FUNCTION_BLOCK "SendRcv_iJaw_1TE"   // FB4, SCL
TITLE = SendRcv_iJaw
{ S7_Optimized_Access := 'TRUE' }
AUTHOR : HeitecAg
VERSION : 0.1
// Kommunikation mit den iJaw Backen mittels IO-LInk und Profinet
   VAR_INPUT
      iLADDR_TigoMaster : HW_DEVICE;   // HW-Device aus Hardwarekonfiguration TigoMaster
      iPN_Act : Bool;   // De-/Aktivierung Profinetteilnehmer 1= Aktivieren 0= Deaktivieren
      iCpuRestart : Bool;   // Restartmerker der SPS Wenn keiner vorhanden dann mit False besetzten.
      iAck_Fehler_IoLinkKom : Bool;   // Quitterung des Kommunikationsfehlers.(Sende-/ Lese Aufträge werden danach erneut gestartet)
      iResetIoLinkKom : Bool;   // Reset der LIO-Link kommunikation (Alle Sende-/ Lese Aufträge werden gelöscht)
      iTime_PnIoRyd : Time;   // Zeit zum Hochlauf des Bussystems / des TigoMasters (Vermeidung von Lesefehlern)
      iIJawAktiv_iJaw1 : Bool;   // iJaw 1 ist aktiv & vorhanden
      iIJawAktiv_iJaw2 : Bool;   // iJaw 2 ist aktiv & vorhanden
      iIJawAktiv_iJaw3 : Bool;   // iJaw 3 ist aktiv & vorhanden
      iIJawAktiv_iJaw4 : Bool;   // iJaw 4 ist aktiv & vorhanden
      iFreeIsduCmd : "UDT_iJawISDUCmdData";   // Freier ISDU-Auftrag
      iFreeIsduSendData : Array[0..#LAENGE_IOLINK_RECORD] of Byte;   // Datenbereich zum Schreiben für den freien ISDU-Auftrag
      iUserDaten_iJaw1 : "UDT_iJawDataSendUser";   // Sendedaten PLC --> iJaw 01
      iUserDaten_iJaw2 : "UDT_iJawDataSendUser";   // Sendedaten PLC --> iJaw 02
      iUserDaten_iJaw3 : "UDT_iJawDataSendUser";   // Sendedaten PLC --> iJaw 03
      iUserDaten_iJaw4 : "UDT_iJawDataSendUser";   // Sendedaten PLC --> iJaw 04
   END_VAR
   VAR_OUTPUT
      oError : Bool;   // Fehler bei der Abarbeitung des Bausteines
      oPnTeilAkt : Bool;   // Status des Profinetteilnehmer 1= Teilnehmer aktiv 0= Teilnehmer deaktiviert
      oIoLinkRdy : Bool;   // Ío link kommunikation bereit zum senden / empfangen
      oIoLinkBusy : Bool;   // Ío link kommunikation beschäftig
      oIoLinkError : Bool;   // Ío link kommunikation fehlerhaft
      oFreeIsduCmdFertig : Bool;   // Freier ISDU-Auftrag erfolgreich abgeschlossen
      oFreeIsduCmdDataBereit : Bool;   // Empfange ISDU-Daten liegen bereit
      oFreeIsduRcvData : Array[0..#LAENGE_IOLINK_RECORD] of Byte;   // Empfange ISDU-Daten
      oUserDaten_iJaw1 : "UDT_iJawDataRcvUser";   // Empfangsdaten PLC <-- iJaw 01
      oUserDaten_iJaw2 : "UDT_iJawDataRcvUser";   // Empfangsdaten PLC <-- iJaw 02
      oUserDaten_iJaw3 : "UDT_iJawDataRcvUser";   // Empfangsdaten PLC <-- iJaw 03
      oUserDaten_iJaw4 : "UDT_iJawDataRcvUser";   // Empfangsdaten PLC <-- iJaw 04
   END_VAR
   VAR
      xlocalInit : Bool := TRUE;   // lokale initalisierung
      xlocalError : Bool;   // lokale Fehler ist aufgetreten
      xMin1iJawVorh : Bool;   // mindesten eine iJaw konfiguriert
      xSchrittketteTimeOut : Bool;   // schrittkette hat ein timeout fehler
      xSchrittErsterZyklus : Bool;   // flanke erster zyklus im schritt
      xFehlerSchrittZeitUeberwachung : Bool;   // fehler schrittzeitüberwachung
      xlocalIoLinkRdy : Bool;   // Ío link kommunikation bereit zum senden / empfangen
      xlocalIoLinkBusy : Bool;   // Ío link kommunikation beschäftig
      xlocalIoLinkError : Bool;   // Ío link kommunikation fehlerhaft
      xlocalFreeIsduCmdFertig : Bool;   // Freier ISDU-Auftrag erfolgreich abgeschlossen
      xlocalFreeIsduCmdDataBereit : Bool;   // Empfange ISDU-Daten liegen bereit
      dtCpuSystemDatumZeit : Date_And_Time;   // datum und uhrzeit cpu
      todCpuSystemZeit : Time_Of_Day;   // zeit des tages cpu
      tSchrittZeitVortag : Time;   // schrittzeit vom vortag
      tCpuSystemZeit : Time;   // zeit der cpu
      tStartZeitSchritt : Time;   // startzeit des aktuellen schrittes
      tAktuelleSchrittzeit : Time;   // aktuelle schrittzeit
      tMinSchrittZeit : Time;   // minimum zeit des aktiven schrittes
      tMaxSchrittZeit : Time;   // maximum zeit des aktiven schrittes (T#0ms = schrittzeit überwachung deaktiviert)
      fpCpuRestart : R_TRIG;   // flanke positiv cpu wurde neugestartet
      fpResetIoLink : R_TRIG;   // flanke positiv trigger reset io-link kommunikation / löschen desfifo puffers
      fpPnIOAktiv : R_TRIG;   // flanke positiv profinetteilnehmer ist aktiviert
      fpPnIOInAktiv : R_TRIG;   // flanke positiv profinetteilnehmer ist deaktiviert
      arrIJawVorhandenAktiv : Array[1..#MAX_ANZAHL_IJAWS] of Bool;   // speicher der überprüfung von vorhandenen und aktiven iJaws
      iRetRcvData : Int;   // retval Profinetdaten lesen
      iRetSer : Int;   // retval Profinetdaten umladen
      iRetSendData : Int;   // retval Profinetdaten schreiben
      iRetValCpuZeitLesen : Int;   // rückgabewert lesen der cpu zeit
      iRetValLog2Geo : Int;   // rückgabewert LOG2GEO
      iRetValWriteBig : Int;   // rückgabewert WRITE_BIG
      iRetValGeoLog : Array[1..#MAX_HW_SLOTS] of Int;   // rückgabewert GEO_LOG
      diAkuelleSchrittnr : DInt := 0;   // aktuelle Schrittnummer
      diAlteSchrittnr : DInt;   // alte Schrittnummer
      diUrAlteSchrittnr : DInt;   // uralte Schrittnummer
      usiLetzterFiFoEintrag : USInt;   // speicher des letzten eintrags im FIFO-Puffer
      tonPNHochlaufzeit : TON_TIME;   // verzögerung profinet hochlaufzeit
      strcDeaktAkt : Struct   // speicher an/abmelden profinet teilnehmer
         ReqAkt : Bool;
         ReqDeak : Bool;
         IstAkt : Bool;
         IstDeak : Bool;
         ModNr : USInt;
         busy : Bool;
         Ret_Val : Int;
         ChangeRequest_old : Bool;
         FP_Changerequest : Bool;
      END_STRUCT;
      strcIoLinkSignale : Struct   // io-link device variablen
         in : Struct
            execute : Bool;   // Anforderung zum Ausführen der Funktion
            hwID : HW_IO;   // Hardware-Kennung des IO-Link-Mastermoduls (Submodul für ET 200eco PN)
            cap : Int;   // Client Access Point (CAP); 0xB400 für ET 200eco PN, CM 8x IO-Link, sonst 0xE003 (227)
            readWrite : Bool;   // FALSE: lesen, TRUE: schreiben
            port : Int;   // Port am IO-Link-Master-Modul
            index : Int;   // Adressparameterindex (IO-Link Device); 0..32767: IOL-D; 65535: Portfunktionen
            subindex : Int;   // Adressparameter Subindex (IO-Link Device); 0: vollständige Aufzeichnung; 1-255: Einzelparameter
            writeLen : Int;   // Länge der Schreibdaten (Nettodaten); 1..232
            timeout : Time := T#20S;   // Zeit, nach der die Anfrage abgebrochen wird
            pollingPeriod : Time := T#100MS;
         END_STRUCT;
         out : Struct
            done : Bool;   // TRUE: FB-Bearbeitung erfolgreich abgeschlossen
            busy : Bool;   // TRUE: FB ist aktiv und neue Ausgangswerte sind zu erwarten.
            error : Bool;   // FALSE: Kein Fehler / TRUE: Bei der Ausführung des FB ist ein Fehler aufgetreten.
            status : Word;   // 16#0000-16#7FFF: Status des FB / 16#8000-16#FFFF: Fehleridentifikation (siehe folgende Tabelle)
            diagnostics : "LIOLink_typeDiagnostics";   // Diagnoseinformationen der FB
            readLen : Int;   // Länge des gelesenen Datensatzes (Anzahl Bytes)
         END_STRUCT;
         record : Array[0..#LAENGE_IOLINK_RECORD] of Byte;   // Datenbereich zum Lesen/Schreiben von Daten (max. 232 Byte)
      END_STRUCT;
      wErrorW0 : Word;   // fehler status io-link device word 0
      wErrorW1 : Word;   // fehler status io-link device word 1
      instLIOLinkDev : "LIOLink_Device";
      fpTriggerFreeISDU : R_TRIG;   // flanken positiv trigger io-link freier isdu auftrag
      fpTriggerTara : Array[1..#MAX_ANZAHL_IJAWS] of R_TRIG;   // flanken positiv trigger io-link kommando tara
      fpTriggerSySMode : Array[1..#MAX_ANZAHL_IJAWS] of R_TRIG;   // flanken positiv trigger io-link kommando sys-mode
      fpTriggerReadType : Array[1..#MAX_ANZAHL_IJAWS] of R_TRIG;   // flanken positiv trigger io-link kommando sys-mode
      fpTriggerIMA : Array[1..#MAX_ANZAHL_IJAWS] of R_TRIG;   // flanken positiv trigger io-link kommando sys-mode
      fpTriggerForceThreshold : Array[1..#MAX_ANZAHL_IJAWS] of R_TRIG;   // flanken positiv trigger io-link kommando sys-mode
      fpTriggerNoiseLevel : Array[1..#MAX_ANZAHL_IJAWS] of R_TRIG;   // flanken positiv trigger io-link kommando sys-mode
      fpTriggerStoreToFlash : Array[1..#MAX_ANZAHL_IJAWS] of R_TRIG;   // flanken positiv trigger io-link kommando sys-mode
      fifoPuffer : Array[1..#MAX_FIFO_IDX] of "UDT_iJawIOFifo";   // fifo-puffer
      hwAnySubSlotsTigoMaster2Th : Array[1..#MAX_HW_SLOTS] of HW_ANY;   // hardware subslot informationen tigomaster 2th
      strIJawType : Array[1..#MAX_ANZAHL_IJAWS] of String;   // Typ des gewähle iJaws
      recordDataFreeISDU : Array[0..#LAENGE_IOLINK_RECORD] of Byte;   // Datenbereich zum Lesen/Schreiben von Daten (max. 232 Byte)
   END_VAR
   VAR_TEMP
      txFPCpuHochlauf : Bool;   // flanke cpu hochlauf / init
      txAktNächstenSchritt : Bool;   // aktiviere nächsten schritt
      tdiI : DInt;   // iterator
      tdiO : DInt;   // iterator
      tempPosSer : DInt;   // pos für de-/serialize
      tempSchrittNr : DInt;   // nächste schrittnummer
      tempHwAny : HW_ANY;   // temporärer hw any
      tempInitRecord : Array[0..#LAENGE_IOLINK_RECORD] of Byte;   // ablesen die Recordaten
      tempHwInfoTigoMaster2Th : GEOADDR;   // hardware slot informationen tigomaster 2th
      tempResetFifo : "UDT_iJawIOFifo";   // reset fifo eintrag
      tempRcvUserdaten : Array[1..#MAX_ANZAHL_IJAWS] of "UDT_iJawDataRcvUser";   // temporär empfangene user-daten
      tempSendUserDaten : Array[1..#MAX_ANZAHL_IJAWS] of "UDT_iJawDataSendUser";   // temporäre user-sende daten
      tempSendDaten : "UDT_iJawDataSend";   // temporär empfangene daten aller iJaw's
      tempRcvEinzelDaten : "UDT_iJawDataRcv";   // temporär empfangene daten einer iJaw
      tempRcvRohDaten : Array[1..#LAENGE_RCV_DATEN] of Byte;   // temporär empfangene roh daten einer iJaw
      tempIJawAktiv : Array[1..#MAX_ANZAHL_IJAWS] of Bool;   // speicher der überprüfung von aktiven iJaws
   END_VAR
   VAR CONSTANT
      MAX_ANZAHL_IJAWS : USInt := 4;   // maximale anzahl von ijaws
      LAENGE_RCV_DATEN : DInt := 33;   // länge von empfangsdaten
      LAENGE_SEND_DATEN : DInt;   // länge von sende daten
      LAENGE_IOLINK_RECORD : DInt := 231;   // länge von io-link record daten
      CAP_IOLINK : Int := 16#B400;   // Client Access Point (CAP); 0xB400 für ET 200eco PN, CM 8x IO-Link, sonst 0xE003 (227)
      CMD_IDLE : USInt := 0;   // kein kommando steht an
      CMD_TARA : USInt := 1;   // Kommando send tara
      CMD_CHANGE_SYSMODE : USInt := 2;   // Kommando send change system mode
      CMD_READ_TYPE : USInt := 3;   // Kommando send read iJaw type
      CMD_APPLICATION_IMA : USInt := 4;   // Kommando send app ima
      CMD_FORCE_TRESHOLD : USInt := 5;   // Kommando send force treshshold
      CMD_NOISE_LEVEL : USInt := 6;   // Kommando send noise level
      CMD_STORE_TO_FLASH : USInt := 7;   // Kommando send strore to flash
      CMD_FREE_ISDU : USInt := 8;   // Kommando freier isdu auftrag
      IDX_CMD_TARA : Int := 518;   // io-link idx cmd tara
      IDX_CMD_SYSMODE : Int := 518;   // io-link idx cmd system mode
      IDX_CMD_READ_TYPE : Int := 518;   // io-link idx cmd system mode
      IDX_CMD_APPLICATION_IMA : Int := 518;   // io-link idx cmd application IMA
      IDX_CMD_FORCE_THRESHOLD : Int := 516;   // io_link idx cmd force treshold
      IDX_CMD_NOISE_LEVEL : Int := 518;   // io_link idx cmd noise level
      IDX_CMD_STORE_TO_FLASH : Int := 517;   // io_link idx cmd store to flash
      SUB_IDX_CMD_TARA : Int := 15;   // io-link sub idx cmd tara
      SUB_IDX_CMD_SYSMODE : USInt := 4;   // io-link sub idx cmd system mode
      SUB_IDX_CMD_READ_TYPE : USInt := 9;   // io-link sub idx cmd read type
      SUB_IDX_CMD_APPLICATION_IMA : Int := 12;   // io-link sub idx cmd application IMA
      SUB_IDX_CMD_FORCE_TRESHOLD : Int := 1;   // io-link sub idx cmd force treshold
      SUB_IDX_CMD_NOISE_LEVEL : Int := 11;   // io-link sub idx cmd noise level
      SUB_IDX_SCMD_TORE_TO_FLASH : Int := 1;   // io-link sub idx store to flash
      RECORD_DATA_TARA : Byte := 1;   // io-link reocrd daten tara
      RECORD_STORE_TO_FLASH : Byte := 1;   // io-link reocrd daten store to flash
      READ : Bool := FALSE;   // io-link Daten lesen
      WRITE : Bool := TRUE;   // io-link Daten schreiben
      SCHRITT_RESET : DInt := 0;   // schrittnummer check io-link kommuikations
      SCHRITT_CHECK_RDY : DInt := 1;   // schrittnummer check io-link kommuikations
      SCHRITT_HOME : DInt := 2;   // schrittnummer home / warte auf befehel
      SCHRITT_SEND_CMD : DInt := 3;   // schrittnummer sende tara
      SCHRITT_WARTE_AUF_DONE : DInt := 11;   // schrittnummer warte auf auftrag abgeschlossen
      SCHRITT_BEARBEITE_FIFO : DInt := 12;   // schrittnummer bearbeite fifo-puffer
      SCHRITT_FEHLER : DInt := 13;   // schrittnummer fehler
      MAX_FIFO_IDX : USInt := 255;   // maximale fifo einträge
      DEF_TIME_OF_DAY : Time_Of_Day := TOD#00:00:00;   // tages start zeit
      MAX_TIME : Time := T#+24d_20h_31m;   // maximal zeit im timeformat
      IDX_FIFO_LESE_INDEX : USInt := 1;   // index des fifo eintrags zum lesen des auftrags
      DEAK_SCHRITT_ZEIT_UEBERW : Time := T#0ms;   // deaktivierung der schrittzeit überwachung
      MAX_HW_SLOTS : DInt := 9;   // maximal slots in hw (8 ijwas + io-link master)
      KEIN_FEHLER : Int := 0;   // kein fehler aufgetreten
      DEF_HW_ANY : HW_ANY := 0;   // default hw any wert
      SLOT_IDX_MAIN_MODUL_2TH : Int := 1;   // hw slot index des 16 port io-link wirles masters
      HW_IDX_IO_LINK_MASTER : Int := 1;   // array index vom io link master
      HW_IDX_IJAW_1 : Int := 2;   // array index von ijaw 1
      HW_IDX_IJAW_2 : Int := 3;   // array index von ijaw 2
      HW_IDX_IJAW_3 : Int := 4;   // array index von ijaw 3
      HW_IDX_IJAW_4 : Int := 5;   // array index von ijaw 4
      LEER_STRING : String;   // leere string zum ablöchen
      CNT_CONV_STRING : UInt := 128;   // Anzahl der zu kopierenden Zeichen. Bei "0" werden alle Zeichen kopiert.
      P_CHAR_CONV_STRING : DInt := 0;   // Position im Array of (W)CHAR / BYTE / WORD, ab der die Zeichen kopiert werden.
   END_VAR
   // // iFreeIsduCmd.port : Port am IO-Link-Master-Modul (Nummer der iJaw 1-8)
BEGIN
   REGION BLOCK INFO HEADER
     //==========================================================================================================
     //Title:        SendRcv_iJaw
     //Function:     Kommunikation mit den iJaw Backen mittels IO-LInk und Profinet (1TE)
     //----------------------------------------------------------------------------------------------------------
     //Change log table:
     //Version       | Date          | Expert in charge      | Changes applied
     //----------------------------------------------------------------------------------------------------------
     //1.0.0         | 15.11.23      | HeitecAg                | First released Version
     //==========================================================================================================
   END_REGION BLOCK INFO HEADER


   REGION INIT

     #xlocalError := FALSE;
     #xSchrittketteTimeOut := FALSE;
     #fpCpuRestart(CLK := #iCpuRestart);

     //Sende Daten vom Bausteineingang einlesen
     #tempSendUserDaten[1] := #iUserDaten_iJaw1;
     #tempSendUserDaten[2] := #iUserDaten_iJaw2;
     #tempSendUserDaten[3] := #iUserDaten_iJaw3;
     #tempSendUserDaten[4] := #iUserDaten_iJaw4;

     //Flanke CPU Hochlauf
     IF #fpCpuRestart.Q
       OR #xlocalInit THEN
       #txFPCpuHochlauf := True;
       #xlocalInit := FALSE;
     ELSE
       #txFPCpuHochlauf := False;
     END_IF;



     //Überbrückung Hochlaufzeit Profinet
     #tonPNHochlaufzeit(IN := TRUE,
                        PT := #iTime_PnIoRyd);

     IF #txFPCpuHochlauf THEN

       #xlocalIoLinkRdy :=
       #xlocalIoLinkBusy :=
       #xlocalIoLinkError :=
       #xlocalFreeIsduCmdFertig :=
       #xlocalFreeIsduCmdDataBereit := FALSE;

       #iRetValLog2Geo := LOG2GEO(LADDR := #iLADDR_TigoMaster, GEOADDR := #tempHwInfoTigoMaster2Th);


       IF #iRetValLog2Geo = 0 THEN
         FOR #tdiI := 1 TO #MAX_HW_SLOTS DO

           #iRetValGeoLog[#tdiI] := GEO_LOG(MASTER := UINT_TO_INT(#tempHwInfoTigoMaster2Th.IOSYSTEM),
                                            STATION := UINT_TO_INT(#tempHwInfoTigoMaster2Th.STATION),
                                            SLOT := #SLOT_IDX_MAIN_MODUL_2TH,
                                            SUBSLOT := DINT_TO_INT(#tdiI),
                                            LADDR => #tempHwAny);

           IF (#iRetValGeoLog[#tdiI] = #KEIN_FEHLER)
             AND (#tempHwAny <> #DEF_HW_ANY) THEN
             #hwAnySubSlotsTigoMaster2Th[#tdiI] := #tempHwAny;
           ELSE
             #hwAnySubSlotsTigoMaster2Th[#tdiI] := #DEF_HW_ANY;
           END_IF;

         END_FOR;
       END_IF;

       #strIJawType[1] := #LEER_STRING;

       FOR #tdiI := 1 TO USINT_TO_DINT(#MAX_ANZAHL_IJAWS) DO
         #strIJawType[#tdiI] := #LEER_STRING;
         ;
       END_FOR;

     END_IF;

     #tempIJawAktiv[1] := #iIJawAktiv_iJaw1;
     #tempIJawAktiv[2] := #iIJawAktiv_iJaw2;
     #tempIJawAktiv[3] := #iIJawAktiv_iJaw3;
     #tempIJawAktiv[4] := #iIJawAktiv_iJaw4;

     REGION CHECK iJAW vorhanden

       #xMin1iJawVorh := FALSE;
       FOR #tdiI := 1 TO USINT_TO_DINT(#MAX_ANZAHL_IJAWS) DO

         IF #tempIJawAktiv[#tdiI]
           AND (#hwAnySubSlotsTigoMaster2Th[#tdiI] <> 0) THEN
           #arrIJawVorhandenAktiv[#tdiI] := TRUE;
           //Mindestens 1 iJaw vorhanden
           #xMin1iJawVorh := TRUE;
         ELSE
           #arrIJawVorhandenAktiv[#tdiI] := FALSE;
         END_IF;

       END_FOR;
     END_REGION CHECK iJAW vorhanden    

   END_REGION INIT

   REGION Profinet Slave aktivieren / deaktivieren
     //Reset bei Hochlauf
     IF #txFPCpuHochlauf THEN
       #strcDeaktAkt.ReqAkt := 0;
       #strcDeaktAkt.ReqDeak := 0;
       #strcDeaktAkt.IstAkt := 0;
       #strcDeaktAkt.IstDeak := 0;
       #strcDeaktAkt.ModNr := 0;
     END_IF;

     //Request PN Slave aktivieren
     IF #tonPNHochlaufzeit.Q AND #iPN_Act AND #xMin1iJawVorh AND NOT #txFPCpuHochlauf AND NOT #strcDeaktAkt.IstAkt THEN
       #strcDeaktAkt.ModNr := 1;
       #strcDeaktAkt.ReqAkt := TRUE;


     END_IF;

     //Request PN Slave deaktivieren
     IF #tonPNHochlaufzeit.Q AND (NOT #iPN_Act OR NOT #xMin1iJawVorh) AND NOT #txFPCpuHochlauf AND NOT #strcDeaktAkt.IstDeak THEN
       #strcDeaktAkt.ModNr := 2;
       #strcDeaktAkt.ReqDeak := TRUE;
       FOR #tdiI := 1 TO USINT_TO_DINT(#MAX_ANZAHL_IJAWS) DO
         #strIJawType[#tdiI] := #LEER_STRING;
         ;
       END_FOR;
     END_IF;

     #fpPnIOAktiv(CLK := #strcDeaktAkt.IstAkt);
     #fpPnIOInAktiv(CLK := #strcDeaktAkt.IstDeak);


     //Teilnehmer aktivieren / deaktivieren
     #strcDeaktAkt.Ret_Val := D_ACT_DP(REQ := #strcDeaktAkt.ReqAkt OR #strcDeaktAkt.ReqDeak, MODE := #strcDeaktAkt.ModNr, LADDR := #iLADDR_TigoMaster, BUSY => #strcDeaktAkt.busy);
     IF (#strcDeaktAkt.Ret_Val = 16#8090)
       OR (#strcDeaktAkt.Ret_Val = 16#8093)
       OR (#strcDeaktAkt.Ret_Val = 16#80a0)
       OR (#strcDeaktAkt.Ret_Val = 16#80a3)
       OR (#strcDeaktAkt.Ret_Val = 16#80a4)
       OR (#strcDeaktAkt.Ret_Val = 16#80c3)
     THEN
       #xlocalError := TRUE;
     END_IF;
     //Zustand Aktiviert / deaktiviert speichern
     //Trigger generieren
     IF #strcDeaktAkt.Ret_Val = 0 AND #strcDeaktAkt.ModNr <> 0 AND NOT #strcDeaktAkt.ChangeRequest_old THEN
       #strcDeaktAkt.FP_Changerequest := True;
     ELSE
       #strcDeaktAkt.FP_Changerequest := false;
     END_IF;
     #strcDeaktAkt.ChangeRequest_old := #strcDeaktAkt.Ret_Val = 0 AND #strcDeaktAkt.ModNr <> 0;

     //Status speicher
     //Slave ist aktiviert
     IF #strcDeaktAkt.FP_Changerequest AND #strcDeaktAkt.ModNr = 1 THEN
       #strcDeaktAkt.ReqAkt := 0;
       #strcDeaktAkt.ReqDeak := 0;
       #strcDeaktAkt.IstAkt := 1;
       #strcDeaktAkt.IstDeak := 0;
       #strcDeaktAkt.ModNr := 0;
       //Slave ist deaktiviert
     ELSIF #strcDeaktAkt.FP_Changerequest AND #strcDeaktAkt.ModNr = 2 THEN
       #strcDeaktAkt.ReqAkt := 0;
       #strcDeaktAkt.ReqDeak := 0;
       #strcDeaktAkt.IstAkt := 0;
       #strcDeaktAkt.IstDeak := 1;
       #strcDeaktAkt.ModNr := 0;
     END_IF;
   END_REGION

   REGION Daten Empfangen
     //Recive Data from iJaws 1..Anzahl iJaws
     //
     IF #xMin1iJawVorh AND #strcDeaktAkt.IstAkt THEN
       FOR #tdiI := 1 TO USINT_TO_DINT(#MAX_ANZAHL_IJAWS) DO

         IF (NOT #arrIJawVorhandenAktiv[#tdiI]) THEN
           CONTINUE;
         END_IF;

         //Empfangsbereich ablöschen
         FOR #tdiO := 1 TO #LAENGE_RCV_DATEN DO
           #tempRcvRohDaten[#tdiO] := 0;
         END_FOR;

         //Daten abholen wenn iJaw N vorhanden
         #iRetRcvData := DPRD_DAT(LADDR := #hwAnySubSlotsTigoMaster2Th[#tdiI + #HW_IDX_IO_LINK_MASTER], RECORD => #tempRcvRohDaten);
         IF #iRetRcvData <> 0 THEN
           #xlocalError := TRUE;
         END_IF;

         //Empfangene Daten aufbereiten
         #tempPosSer := 0;
         #iRetSer := Deserialize(SRC_ARRAY := #tempRcvRohDaten, DEST_VARIABLE => #tempRcvEinzelDaten, POS := #tempPosSer);
         IF #iRetSer <> 0 THEN
           #xlocalError := TRUE;
         END_IF;

         #tempRcvUserdaten[#tdiI].Gauge1 := WORD_TO_UINT(#tempRcvEinzelDaten.Gauge1);
         #tempRcvUserdaten[#tdiI].Gauge2 := WORD_TO_UINT(#tempRcvEinzelDaten.Gauge2);
         #tempRcvUserdaten[#tdiI].Battery := BYTE_TO_USINT(#tempRcvEinzelDaten.Battery);
         #tempRcvUserdaten[#tdiI].Temperature := BYTE_TO_SINT(#tempRcvEinzelDaten.Temperature);
         #tempRcvUserdaten[#tdiI].GyroXaxis := BYTE_TO_SINT(#tempRcvEinzelDaten.GyroXaxis);
         #tempRcvUserdaten[#tdiI].GyroYaxis := BYTE_TO_SINT(#tempRcvEinzelDaten.GyroYaxis);
         #tempRcvUserdaten[#tdiI].GyroZaxis := BYTE_TO_SINT(#tempRcvEinzelDaten.GyroZaxis);
         #tempRcvUserdaten[#tdiI].Force1 := WORD_TO_UINT(#tempRcvEinzelDaten.Force1);
         #tempRcvUserdaten[#tdiI].Force2 := WORD_TO_UINT(#tempRcvEinzelDaten.Force2);
       END_FOR;

     END_IF;

     #tempRcvUserdaten[1].iJawType := #strIJawType[1];
     #tempRcvUserdaten[2].iJawType := #strIJawType[2];
     #tempRcvUserdaten[3].iJawType := #strIJawType[3];
     #tempRcvUserdaten[4].iJawType := #strIJawType[4];


     //Empfangene Daten auf Bausteinausgang schreiben
     #oUserDaten_iJaw1 := #tempRcvUserdaten[1];
     #oUserDaten_iJaw2 := #tempRcvUserdaten[2];
     #oUserDaten_iJaw3 := #tempRcvUserdaten[3];
     #oUserDaten_iJaw4 := #tempRcvUserdaten[4];

   END_REGION

   REGION RESET FIFO PUFFER
     #fpResetIoLink(CLK := #iResetIoLinkKom);

     IF #txFPCpuHochlauf
       OR #fpResetIoLink.Q
       OR #fpPnIOAktiv.Q
       OR #fpPnIOInAktiv.Q
     THEN
       FOR #tdiI := 1 TO USINT_TO_DINT(#MAX_FIFO_IDX) DO
         #fifoPuffer[#tdiI] := #tempResetFifo;
         #usiLetzterFiFoEintrag := 0;
         #diAkuelleSchrittnr := #SCHRITT_RESET;
       END_FOR;
     END_IF;
   END_REGION RESET FIFO PUFFER

   REGION FIFO PUFFER IO-LINK KOMMANDOS
     IF #xMin1iJawVorh AND #strcDeaktAkt.IstAkt THEN

       #fpTriggerFreeISDU(CLK := #iFreeIsduCmd.execute);


       FOR #tdiI := 1 TO USINT_TO_DINT(#MAX_ANZAHL_IJAWS) DO

         #fpTriggerTara[#tdiI](CLK := #tempSendUserDaten[#tdiI].RelCmdTara);
         #fpTriggerSySMode[#tdiI](CLK := #tempSendUserDaten[#tdiI].RelCmdSysMode);
         #fpTriggerReadType[#tdiI](CLK := #tempSendUserDaten[#tdiI].RelReadType);
         #fpTriggerIMA[#tdiI](CLK := #tempSendUserDaten[#tdiI].RelIMA);
         #fpTriggerForceThreshold[#tdiI](CLK := #tempSendUserDaten[#tdiI].RelForceTreshold);
         #fpTriggerNoiseLevel[#tdiI](CLK := #tempSendUserDaten[#tdiI].RelNoiseLevel);
         #fpTriggerStoreToFlash[#tdiI](CLK := #tempSendUserDaten[#tdiI].RelStoreToFlash);




         IF #fpTriggerTara[#tdiI].Q AND #arrIJawVorhandenAktiv[#tdiI] THEN

           #usiLetzterFiFoEintrag += 1;
           #fifoPuffer[#usiLetzterFiFoEintrag].cmd := #CMD_TARA;
           #fifoPuffer[#usiLetzterFiFoEintrag].isuCmdData.execute := TRUE;
           #fifoPuffer[#usiLetzterFiFoEintrag].isuCmdData.readWrite := #WRITE;
           #fifoPuffer[#usiLetzterFiFoEintrag].isuCmdData."port" := DINT_TO_INT(#tdiI);
           #fifoPuffer[#usiLetzterFiFoEintrag].isuCmdData.index := #IDX_CMD_TARA;
           #fifoPuffer[#usiLetzterFiFoEintrag].isuCmdData.subindex := #SUB_IDX_CMD_TARA;
           #fifoPuffer[#usiLetzterFiFoEintrag].isuCmdData.writeLen := 1;

         END_IF;

         IF #fpTriggerSySMode[#tdiI].Q AND #arrIJawVorhandenAktiv[#tdiI] THEN
           #usiLetzterFiFoEintrag += 1;
           #fifoPuffer[#usiLetzterFiFoEintrag].cmd := #CMD_CHANGE_SYSMODE;
           #fifoPuffer[#usiLetzterFiFoEintrag].isuCmdData.execute := TRUE;
           #fifoPuffer[#usiLetzterFiFoEintrag].isuCmdData.readWrite := #WRITE;
           #fifoPuffer[#usiLetzterFiFoEintrag].isuCmdData."port" := DINT_TO_INT(#tdiI);
           #fifoPuffer[#usiLetzterFiFoEintrag].isuCmdData.index := #IDX_CMD_SYSMODE;
           #fifoPuffer[#usiLetzterFiFoEintrag].isuCmdData.subindex := #SUB_IDX_CMD_SYSMODE;
           #fifoPuffer[#usiLetzterFiFoEintrag].isuCmdData.writeLen := 1;
         END_IF;

         IF #fpTriggerReadType[#tdiI].Q AND #arrIJawVorhandenAktiv[#tdiI] THEN
           #usiLetzterFiFoEintrag += 1;
           #fifoPuffer[#usiLetzterFiFoEintrag].cmd := #CMD_READ_TYPE;
           #fifoPuffer[#usiLetzterFiFoEintrag].isuCmdData.execute := TRUE;
           #fifoPuffer[#usiLetzterFiFoEintrag].isuCmdData.readWrite := #READ;
           #fifoPuffer[#usiLetzterFiFoEintrag].isuCmdData."port" := DINT_TO_INT(#tdiI);
           #fifoPuffer[#usiLetzterFiFoEintrag].isuCmdData.index := #IDX_CMD_READ_TYPE;
           #fifoPuffer[#usiLetzterFiFoEintrag].isuCmdData.subindex := #SUB_IDX_CMD_READ_TYPE;
           #fifoPuffer[#usiLetzterFiFoEintrag].isuCmdData.writeLen := 0;
         END_IF;

         IF #fpTriggerIMA[#tdiI].Q AND #arrIJawVorhandenAktiv[#tdiI] THEN
           #usiLetzterFiFoEintrag += 1;
           #fifoPuffer[#usiLetzterFiFoEintrag].cmd := #CMD_APPLICATION_IMA;
           #fifoPuffer[#usiLetzterFiFoEintrag].isuCmdData.execute := TRUE;
           #fifoPuffer[#usiLetzterFiFoEintrag].isuCmdData.readWrite := #WRITE;
           #fifoPuffer[#usiLetzterFiFoEintrag].isuCmdData."port" := DINT_TO_INT(#tdiI);
           #fifoPuffer[#usiLetzterFiFoEintrag].isuCmdData.index := #IDX_CMD_APPLICATION_IMA;
           #fifoPuffer[#usiLetzterFiFoEintrag].isuCmdData.subindex := #SUB_IDX_CMD_APPLICATION_IMA;
           #fifoPuffer[#usiLetzterFiFoEintrag].isuCmdData.writeLen := 1;
         END_IF;

         IF #fpTriggerForceThreshold[#tdiI].Q AND #arrIJawVorhandenAktiv[#tdiI] THEN
           #usiLetzterFiFoEintrag += 1;
           #fifoPuffer[#usiLetzterFiFoEintrag].cmd := #CMD_FORCE_TRESHOLD;
           #fifoPuffer[#usiLetzterFiFoEintrag].isuCmdData.execute := TRUE;
           #fifoPuffer[#usiLetzterFiFoEintrag].isuCmdData.readWrite := #WRITE;
           #fifoPuffer[#usiLetzterFiFoEintrag].isuCmdData."port" := DINT_TO_INT(#tdiI);
           #fifoPuffer[#usiLetzterFiFoEintrag].isuCmdData.index := #IDX_CMD_FORCE_THRESHOLD;
           #fifoPuffer[#usiLetzterFiFoEintrag].isuCmdData.subindex := #SUB_IDX_CMD_FORCE_TRESHOLD;
           #fifoPuffer[#usiLetzterFiFoEintrag].isuCmdData.writeLen := 4;
         END_IF;

         IF #fpTriggerNoiseLevel[#tdiI].Q AND #arrIJawVorhandenAktiv[#tdiI] THEN
           #usiLetzterFiFoEintrag += 1;
           #fifoPuffer[#usiLetzterFiFoEintrag].cmd := #CMD_NOISE_LEVEL;
           #fifoPuffer[#usiLetzterFiFoEintrag].isuCmdData.execute := TRUE;
           #fifoPuffer[#usiLetzterFiFoEintrag].isuCmdData.readWrite := #WRITE;
           #fifoPuffer[#usiLetzterFiFoEintrag].isuCmdData."port" := DINT_TO_INT(#tdiI);
           #fifoPuffer[#usiLetzterFiFoEintrag].isuCmdData.index := #IDX_CMD_NOISE_LEVEL;
           #fifoPuffer[#usiLetzterFiFoEintrag].isuCmdData.subindex := #SUB_IDX_CMD_NOISE_LEVEL;
           #fifoPuffer[#usiLetzterFiFoEintrag].isuCmdData.writeLen := 2;
         END_IF;

         IF #fpTriggerStoreToFlash[#tdiI].Q AND #arrIJawVorhandenAktiv[#tdiI] THEN
           #usiLetzterFiFoEintrag += 1;
           #fifoPuffer[#usiLetzterFiFoEintrag].cmd := #CMD_STORE_TO_FLASH;
           #fifoPuffer[#usiLetzterFiFoEintrag].isuCmdData.execute := TRUE;
           #fifoPuffer[#usiLetzterFiFoEintrag].isuCmdData.readWrite := #WRITE;
           #fifoPuffer[#usiLetzterFiFoEintrag].isuCmdData."port" := DINT_TO_INT(#tdiI);
           #fifoPuffer[#usiLetzterFiFoEintrag].isuCmdData.index := #IDX_CMD_STORE_TO_FLASH;
           #fifoPuffer[#usiLetzterFiFoEintrag].isuCmdData.subindex := #SUB_IDX_SCMD_TORE_TO_FLASH;
           #fifoPuffer[#usiLetzterFiFoEintrag].isuCmdData.writeLen := 1;
         END_IF;

         IF #fpTriggerFreeISDU.Q
           AND (#iFreeIsduCmd."port" <=#MAX_ANZAHL_IJAWS)
           AND (#iFreeIsduCmd."port" >= 1)THEN
           IF #arrIJawVorhandenAktiv[#iFreeIsduCmd."port"] THEN
             #usiLetzterFiFoEintrag += 1;
             #fifoPuffer[#usiLetzterFiFoEintrag].cmd := #CMD_FREE_ISDU;
             #fifoPuffer[#usiLetzterFiFoEintrag].isuCmdData.execute := TRUE;
             #fifoPuffer[#usiLetzterFiFoEintrag].isuCmdData.readWrite := #iFreeIsduCmd.readWrite;
             #fifoPuffer[#usiLetzterFiFoEintrag].isuCmdData."port" := #iFreeIsduCmd."port";
             #fifoPuffer[#usiLetzterFiFoEintrag].isuCmdData.index := #iFreeIsduCmd.index;
             #fifoPuffer[#usiLetzterFiFoEintrag].isuCmdData.subindex := #iFreeIsduCmd.subindex;
             #fifoPuffer[#usiLetzterFiFoEintrag].isuCmdData.writeLen := #iFreeIsduCmd.writeLen;

             #xlocalFreeIsduCmdFertig := FALSE;
             #xlocalFreeIsduCmdDataBereit := FALSE;
             #oFreeIsduRcvData := #tempInitRecord;
           END_IF;
         END_IF;

       END_FOR;
     END_IF;
   END_REGION FIFO PUFFER IO-LINK KOMMANDOS

   REGION Schrittkette Kommandos schreiben

     IF #xMin1iJawVorh AND #strcDeaktAkt.IstAkt THEN
       // Statement section REGION
       CASE #diAkuelleSchrittnr OF

         #SCHRITT_RESET:

           (*IO-Link Status setzten*)
           #xlocalIoLinkRdy := FALSE;
           #xlocalIoLinkBusy := FALSE;
           #xlocalIoLinkError := FALSE;

           IF (#hwAnySubSlotsTigoMaster2Th[#HW_IDX_IO_LINK_MASTER] <> #DEF_HW_ANY) THEN
             #tempSchrittNr := #SCHRITT_CHECK_RDY;
             #txAktNächstenSchritt := TRUE;
             #strcIoLinkSignale.in.execute := FALSE;
           END_IF;

         #SCHRITT_CHECK_RDY:

           (*IO-Link Status setzten*)
           #xlocalIoLinkRdy := FALSE;
           #xlocalIoLinkBusy := FALSE;
           #xlocalIoLinkError := FALSE;

           IF (#strcDeaktAkt.IstAkt AND NOT #strcDeaktAkt.IstDeak)
             AND (NOT #strcIoLinkSignale.out.error)
             AND (#strcIoLinkSignale.out.status = 16#7000)
           THEN
             #tempSchrittNr := #SCHRITT_HOME;
             #txAktNächstenSchritt := TRUE;
           ELSIF (#strcIoLinkSignale.out.status = 16#8000)
             OR #strcIoLinkSignale.out.error
             AND (NOT #xSchrittErsterZyklus) THEN
             #tempSchrittNr := #SCHRITT_FEHLER;
             #txAktNächstenSchritt := TRUE;
           END_IF;

         #SCHRITT_HOME:

           (*IO-Link Status setzten*)
           #xlocalIoLinkRdy := TRUE;
           #xlocalIoLinkBusy := FALSE;
           #xlocalIoLinkError := FALSE;

           IF (#fifoPuffer[#IDX_FIFO_LESE_INDEX].cmd = #CMD_IDLE) THEN
             ;
           ELSIF (#fifoPuffer[#IDX_FIFO_LESE_INDEX].cmd = #CMD_TARA) THEN
             #tempSchrittNr := #SCHRITT_SEND_CMD;
             #txAktNächstenSchritt := TRUE;
           ELSIF (#fifoPuffer[#IDX_FIFO_LESE_INDEX].cmd = #CMD_CHANGE_SYSMODE) THEN
             #tempSchrittNr := #SCHRITT_SEND_CMD;
             #txAktNächstenSchritt := TRUE;
           ELSIF (#fifoPuffer[#IDX_FIFO_LESE_INDEX].cmd = #CMD_READ_TYPE) THEN
             #tempSchrittNr := #SCHRITT_SEND_CMD;
             #txAktNächstenSchritt := TRUE;
           ELSIF (#fifoPuffer[#IDX_FIFO_LESE_INDEX].cmd = #CMD_APPLICATION_IMA) THEN
             #tempSchrittNr := #SCHRITT_SEND_CMD;
             #txAktNächstenSchritt := TRUE;
           ELSIF (#fifoPuffer[#IDX_FIFO_LESE_INDEX].cmd = #"CMD_FORCE_TRESHOLD") THEN
             #tempSchrittNr := #SCHRITT_SEND_CMD;
             #txAktNächstenSchritt := TRUE;
           ELSIF (#fifoPuffer[#IDX_FIFO_LESE_INDEX].cmd = #CMD_NOISE_LEVEL) THEN
             #tempSchrittNr := #SCHRITT_SEND_CMD;
             #txAktNächstenSchritt := TRUE;
           ELSIF (#fifoPuffer[#IDX_FIFO_LESE_INDEX].cmd = #CMD_STORE_TO_FLASH) THEN
             #tempSchrittNr := #SCHRITT_SEND_CMD;
           ELSIF (#fifoPuffer[#IDX_FIFO_LESE_INDEX].cmd = #CMD_FREE_ISDU) THEN
             #tempSchrittNr := #SCHRITT_SEND_CMD;
             #txAktNächstenSchritt := TRUE;
           END_IF;

         #SCHRITT_SEND_CMD:

           (*IO-Link Status setzten*)
           #xlocalIoLinkRdy := FALSE;
           #xlocalIoLinkBusy := TRUE;
           #xlocalIoLinkError := FALSE;

           // Reset Record daten
           #strcIoLinkSignale.record := #tempInitRecord;

           #strcIoLinkSignale.in.execute := #fifoPuffer[#IDX_FIFO_LESE_INDEX].isuCmdData.execute;
           #strcIoLinkSignale.in."port" := #fifoPuffer[#IDX_FIFO_LESE_INDEX].isuCmdData."port";
           #strcIoLinkSignale.in.index := #fifoPuffer[#IDX_FIFO_LESE_INDEX].isuCmdData.index;
           #strcIoLinkSignale.in.subindex := #fifoPuffer[#IDX_FIFO_LESE_INDEX].isuCmdData.subindex;
           #strcIoLinkSignale.in.writeLen := #fifoPuffer[#IDX_FIFO_LESE_INDEX].isuCmdData.writeLen;
           #strcIoLinkSignale.in.readWrite := #fifoPuffer[#IDX_FIFO_LESE_INDEX].isuCmdData.readWrite;

           IF (#fifoPuffer[#IDX_FIFO_LESE_INDEX].cmd = #CMD_TARA) THEN
             #strcIoLinkSignale.record[0] := #RECORD_DATA_TARA;

           ELSIF (#fifoPuffer[#IDX_FIFO_LESE_INDEX].cmd = #CMD_CHANGE_SYSMODE) THEN
             #strcIoLinkSignale.record[0] := #tempSendUserDaten[#fifoPuffer[#IDX_FIFO_LESE_INDEX].isuCmdData."port"].Mode;

           ELSIF (#fifoPuffer[#IDX_FIFO_LESE_INDEX].cmd = #CMD_APPLICATION_IMA) THEN
             #strcIoLinkSignale.record[0] := USINT_TO_BYTE(#tempSendUserDaten[#fifoPuffer[#IDX_FIFO_LESE_INDEX].isuCmdData."port"].IMA);

           ELSIF (#fifoPuffer[#IDX_FIFO_LESE_INDEX].cmd = #CMD_FORCE_TRESHOLD) THEN
             #tempPosSer := 0;
             #iRetValWriteBig := WRITE_BIG(src_variable := #tempSendUserDaten[#fifoPuffer[#IDX_FIFO_LESE_INDEX].isuCmdData."port"].ForceTreshold,
                                           dest_array := #strcIoLinkSignale.record,
                                           pos := #tempPosSer);


           ELSIF (#fifoPuffer[#IDX_FIFO_LESE_INDEX].cmd = #CMD_NOISE_LEVEL) THEN
             #tempPosSer := 0;
             #iRetValWriteBig := WRITE_BIG(src_variable := #tempSendUserDaten[#fifoPuffer[#IDX_FIFO_LESE_INDEX].isuCmdData."port"].NoiseLevel,
                                           dest_array := #strcIoLinkSignale.record,
                                           pos := #tempPosSer);

           ELSIF (#fifoPuffer[#IDX_FIFO_LESE_INDEX].cmd = #CMD_STORE_TO_FLASH) THEN
             #strcIoLinkSignale.record[0] := #RECORD_STORE_TO_FLASH;

           ELSIF (#fifoPuffer[#IDX_FIFO_LESE_INDEX].cmd = #CMD_READ_TYPE) THEN
             ;

           ELSIF (#fifoPuffer[#IDX_FIFO_LESE_INDEX].cmd = #CMD_FREE_ISDU) THEN
             #strcIoLinkSignale.record := #iFreeIsduSendData;
           END_IF;

           IF #strcIoLinkSignale.out.error
             OR (#iRetValWriteBig <> 0) THEN
             #tempSchrittNr := #SCHRITT_FEHLER;
             #txAktNächstenSchritt := TRUE;
           ELSIF #strcIoLinkSignale.out.busy
             AND (NOT #strcIoLinkSignale.out.done) THEN
             #tempSchrittNr := #SCHRITT_WARTE_AUF_DONE;
             #txAktNächstenSchritt := TRUE;
           END_IF;

         #SCHRITT_WARTE_AUF_DONE:

           (*IO-Link Status setzten*)
           #xlocalIoLinkRdy := FALSE;
           #xlocalIoLinkBusy := TRUE;
           #xlocalIoLinkError := FALSE;

           IF #strcIoLinkSignale.out.done THEN

             IF (#fifoPuffer[#IDX_FIFO_LESE_INDEX].cmd = #CMD_READ_TYPE) THEN
               Chars_TO_Strg(Chars  := #strcIoLinkSignale.record,
                             pChars := #P_CHAR_CONV_STRING,
                             Cnt    := #CNT_CONV_STRING,
                             Strg   => #strIJawType[#fifoPuffer[#IDX_FIFO_LESE_INDEX].isuCmdData."port"]);

             ELSIF (#fifoPuffer[#IDX_FIFO_LESE_INDEX].cmd = #CMD_FREE_ISDU) THEN

               #xlocalFreeIsduCmdFertig := TRUE;
               #oFreeIsduRcvData := #tempInitRecord;

               IF (#fifoPuffer[#IDX_FIFO_LESE_INDEX].isuCmdData.readWrite = #READ) THEN
                 #xlocalFreeIsduCmdDataBereit := TRUE;
                 #recordDataFreeISDU := #strcIoLinkSignale.record;
               ELSE
                 #xlocalFreeIsduCmdDataBereit := FALSE;
               END_IF;

             END_IF;

             #strcIoLinkSignale.in.execute := FALSE;
             #tempSchrittNr := #SCHRITT_BEARBEITE_FIFO;
             #txAktNächstenSchritt := TRUE;
           ELSIF #strcIoLinkSignale.out.error THEN
             #tempSchrittNr := #SCHRITT_FEHLER;
             #txAktNächstenSchritt := TRUE;
           END_IF;


         #SCHRITT_BEARBEITE_FIFO:

           (*IO-Link Status setzten*)
           #xlocalIoLinkRdy := FALSE;
           #xlocalIoLinkBusy := TRUE;
           #xlocalIoLinkError := FALSE;

           FOR #tdiO := USINT_TO_DINT(#usiLetzterFiFoEintrag) TO 1 BY -1 DO
             IF (#tdiO = 1) THEN
               #fifoPuffer[#tdiO] := #tempResetFifo;
               #usiLetzterFiFoEintrag += -1;
             ELSIF
               (#tdiO <= USINT_TO_DINT(#MAX_FIFO_IDX))
               AND (#tdiO > 1) THEN
               #fifoPuffer[#tdiO - 1] := #fifoPuffer[#tdiO];
               #fifoPuffer[#tdiO] := #tempResetFifo;
               #usiLetzterFiFoEintrag += -1;
             ELSE
               EXIT;
             END_IF;
           END_FOR;

           #tempSchrittNr := #SCHRITT_CHECK_RDY;
           #txAktNächstenSchritt := TRUE;

         #SCHRITT_FEHLER:

           (*IO-Link Status setzten*)
           #xlocalIoLinkRdy := FALSE;
           #xlocalIoLinkBusy := FALSE;
           #xlocalIoLinkError := TRUE;

           #xSchrittketteTimeOut := TRUE;
           #xlocalError := TRUE;

           IF #iAck_Fehler_IoLinkKom THEN

             #strcIoLinkSignale.in.execute := FALSE;

             #tempSchrittNr := #SCHRITT_CHECK_RDY;
             #txAktNächstenSchritt := TRUE;
           END_IF;

         ELSE  // Statement section ELSE
           ;
       END_CASE;

       REGION SCHRITT UMSCHALTUNG
         #xSchrittErsterZyklus := FALSE;

         IF #txAktNächstenSchritt
           AND (#tempSchrittNr >= #SCHRITT_CHECK_RDY)
           AND (#tempSchrittNr <= #SCHRITT_FEHLER) THEN
           #diUrAlteSchrittnr := #diAlteSchrittnr;
           #diAlteSchrittnr := #diAkuelleSchrittnr;
           #diAkuelleSchrittnr := #tempSchrittNr;
           #xSchrittErsterZyklus := TRUE;
         END_IF;

         REGION SCHRITTZEIT
           #iRetValCpuZeitLesen := RD_SYS_T(#dtCpuSystemDatumZeit);
           #todCpuSystemZeit := DT_TO_TOD(#dtCpuSystemDatumZeit);
           #tCpuSystemZeit := TOD_TO_TIME(#todCpuSystemZeit);

           IF #xSchrittErsterZyklus
             OR (#tAktuelleSchrittzeit >= #MAX_TIME) THEN
             #tStartZeitSchritt := #tCpuSystemZeit;
             #tSchrittZeitVortag := #DEAK_SCHRITT_ZEIT_UEBERW;
           ELSIF (#todCpuSystemZeit = #DEF_TIME_OF_DAY) THEN
             #tSchrittZeitVortag := #tAktuelleSchrittzeit;
             #tStartZeitSchritt := #tCpuSystemZeit;
           END_IF;

           #tAktuelleSchrittzeit := (#tCpuSystemZeit - #tStartZeitSchritt) + #tSchrittZeitVortag;

           IF (#tMaxSchrittZeit > #DEAK_SCHRITT_ZEIT_UEBERW)
             AND (#tMaxSchrittZeit > #tAktuelleSchrittzeit)
           THEN
             #xFehlerSchrittZeitUeberwachung := TRUE;
           ELSE
             #xFehlerSchrittZeitUeberwachung := FALSE;
           END_IF;

         END_REGION SCHRITTZEIT


       END_REGION SCHRITT UMSCHALTUNG
     ELSE
       #xlocalIoLinkRdy := FALSE;
       #xlocalIoLinkBusy := FALSE;
       #xlocalIoLinkError := FALSE;

     END_IF;

   END_REGION

   REGION BEREITSTELLUNG RCV DATEN FREE ISDU-AUFTRAG
     IF #iFreeIsduCmd.execute
       AND (#strcDeaktAkt.IstAkt AND NOT #strcDeaktAkt.IstDeak)
     THEN
       IF #xlocalFreeIsduCmdFertig
         AND #xlocalFreeIsduCmdDataBereit
       THEN
         #oFreeIsduRcvData := #recordDataFreeISDU;
       END_IF;
     ELSE
       #xlocalFreeIsduCmdFertig := FALSE;
       #xlocalFreeIsduCmdDataBereit := FALSE;
       #oFreeIsduRcvData := #recordDataFreeISDU := #tempInitRecord;
     END_IF;
   END_REGION BEREITSTELLUNG RCV DATEN FREE ISDU-AUFTRAG


   REGION AUFRUF IO_LINK DEVICE

     REGION INIT IO-Link
       #strcIoLinkSignale.in.hwID := #hwAnySubSlotsTigoMaster2Th[#HW_IDX_IO_LINK_MASTER];
       #strcIoLinkSignale.in.cap := #CAP_IOLINK;
     END_REGION INIT IO-Link 

     #instLIOLinkDev(execute       := #strcIoLinkSignale.in.execute,
                     hwID          := #strcIoLinkSignale.in.hwID,
                     cap           := #strcIoLinkSignale.in.cap,
                     readWrite     := #strcIoLinkSignale.in.readWrite,
                     "port"        := #strcIoLinkSignale.in."port",
                     index         := #strcIoLinkSignale.in.index,
                     subindex      := #strcIoLinkSignale.in.subindex,
                     writeLen      := #strcIoLinkSignale.in.writeLen,
                     timeout       := #strcIoLinkSignale.in.timeout,
                     pollingPeriod := #strcIoLinkSignale.in.pollingPeriod,
                     done          => #strcIoLinkSignale.out.done,
                     busy          => #strcIoLinkSignale.out.busy,
                     error         => #strcIoLinkSignale.out.error,
                     status        => #strcIoLinkSignale.out.status,
                     diagnostics   => #strcIoLinkSignale.out.diagnostics,
                     readLen       => #strcIoLinkSignale.out.readLen,
                     record        := #strcIoLinkSignale.record);

     #wErrorW0 := #strcIoLinkSignale.out.diagnostics.subfunctionStatus.%W0;
     #wErrorW1 := #strcIoLinkSignale.out.diagnostics.subfunctionStatus.%W1;


   END_REGION AUFRUF IO_LINK DEVICE

   REGION Daten senden
     //Daten senden an iJaw 1..Anzahl iJaws

     IF #xMin1iJawVorh AND #strcDeaktAkt.IstAkt THEN

       //Daten aufbereiten
       FOR #tdiI := 1 TO USINT_TO_DINT(#MAX_ANZAHL_IJAWS) DO
         IF (NOT #arrIJawVorhandenAktiv[#tdiI]) THEN
           CONTINUE;
         END_IF;

         //wenn iJaw vorhanden
         #tempSendDaten.nRotSpeedSpindleAct := #tempSendUserDaten[#tdiI].nRotSpeedSpindleAct;
         #tempSendDaten.pHydCylChamber1Act := #tempSendUserDaten[#tdiI].pHydCylChamber1Act;
         #tempSendDaten.pHydCylChamber2Act := #tempSendUserDaten[#tdiI].pHydCylChamber2Act;
         #tempSendDaten.AHydCylChamber1Act := #tempSendUserDaten[#tdiI].AHydCylChamber1Act;
         #tempSendDaten.AHydCylChamber2Act := #tempSendUserDaten[#tdiI].AHydCylChamber2Act;

         //Daten senden
         IF #strcDeaktAkt.IstAkt THEN
           #iRetSendData := DPWR_DAT(LADDR := #hwAnySubSlotsTigoMaster2Th[#tdiI + #HW_IDX_IO_LINK_MASTER], RECORD := #tempSendDaten);
           IF #iRetSendData <> 0 THEN
             #xlocalError := TRUE;
           END_IF;
         END_IF;
       END_FOR;
     END_IF;
   END_REGION

   REGION BAUSTEIN ENDE
     #oIoLinkRdy := #xlocalIoLinkRdy;
     #oIoLinkBusy := #xlocalIoLinkBusy;
     #oIoLinkError := #xlocalIoLinkError;

     #oFreeIsduCmdFertig := #xlocalFreeIsduCmdFertig;
     #oFreeIsduCmdDataBereit := #xlocalFreeIsduCmdDataBereit;

     // Setze Bausteinausgang Teilnehmer aktiv
     #oPnTeilAkt := #strcDeaktAkt.IstAkt AND NOT #strcDeaktAkt.IstDeak;

     #oError := #xlocalError;
     ENO := (NOT #xlocalError);
     RETURN;
   END_REGION BAUSTEIN ENDE
END_FUNCTION_BLOCK

// ===== library: MasterCopy "AufrufSendRcvIJaw" =====

FUNCTION_BLOCK "AufrufSendRcvIJaw"   // FB1, LAD
{ S7_Optimized_Access := 'TRUE' }
VERSION : 0.1
   VAR
      instSendReciJaw8P : "SendRcv_iJaw";
      instSendReciJaw4P : "SendRcv_iJaw_1TE";
      hwDeviceTigoMaster : HW_DEVICE;   // Ermittelte Hardware-Kennung des TigoMasters
      testGain : UInt;
      Fehlerinformation : Int;
   END_VAR
   VAR_TEMP
      tiRetval : Int;   // Rückgabewert / FehlerCode GetHwDevice
      tPos : DInt;
   END_VAR
   VAR CONSTANT
      IDX_IJAW_1 : Int := 1;   // Index der iJaw 1
      IDX_IJAW_2 : Int := 2;   // Index der iJaw 2
      IDX_IJAW_3 : Int := 3;   // Index der iJaw 3
      IDX_IJAW_4 : Int := 4;   // Index der iJaw 4
      IDX_IJAW_5 : Int := 5;   // Index der iJaw 5
      IDX_IJAW_6 : Int := 6;   // Index der iJaw 6
      IDX_IJAW_7 : Int := 7;   // Index der iJaw 7
      IDX_IJAW_8 : Int := 8;   // Index der iJaw 8
      IDX_ISDU_CMD_GAIN : Int := 515;   // ISDU Index des Kommandos Gain
      SUB_IDX_ISDU_CMD_GAIN : Int := 1;   // ISDU Subindex des Kommandos Gain
      READ_WRITE_ISDU_CMD_GAIN : Bool := FALSE;   // ISDU Schreiben / Lesen FALSE: lesen, TRUE: schreiben
      WRITE_LENGTH_ISDU_CMD_GAIN : Int := 2;   // ISDU Länge der Schreibdaten (Nettodaten); 1..232
   END_VAR
   VAR_TEMP   // added for the SCL form of the ladder/FBD networks
      _w1 : Bool;
   END_VAR
BEGIN

REGION Network 1: ERMITTELN DER HW_DEVICE KENNENUNG
   // An varEaAdresse muss eine E/A-Adresse von iJawXX parametriert werden.
   // Wird die Systemkonstante HW_DEVICE vom TigoMaster benutzt kann das Netwerk gelöscht werden.
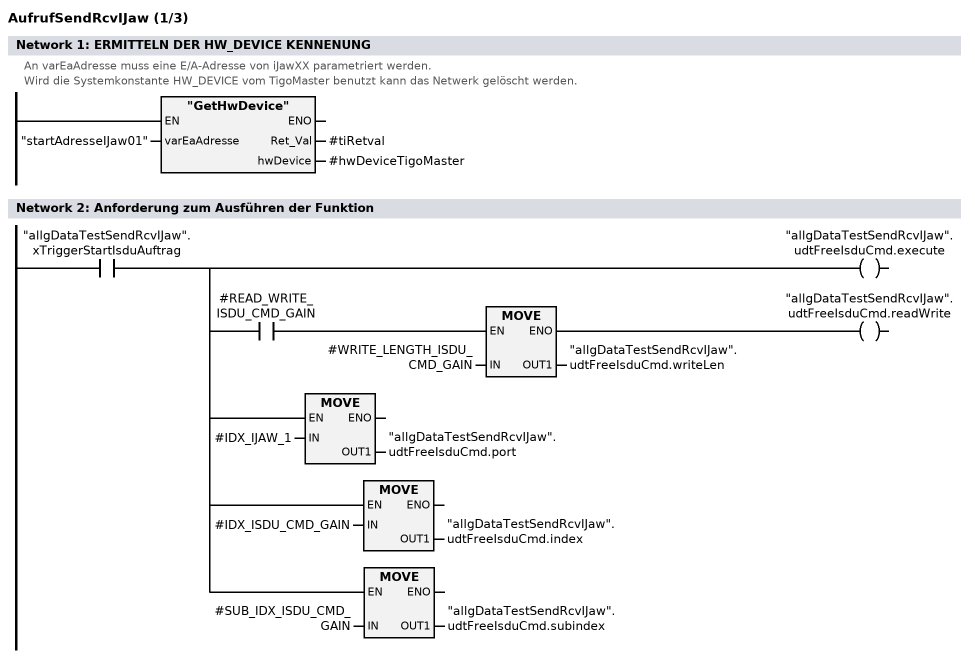
   RUNG wire#powerrail
      "GetHwDevice"(varEaAdresse := "startAdresseIJaw01", Ret_Val => #tiRetval, hwDevice => #hwDeviceTigoMaster)
   END_RUNG
   // the same network as SCL:
   #tiRetval := "GetHwDevice"(varEaAdresse := "startAdresseIJaw01", hwDevice => #hwDeviceTigoMaster);
END_REGION

REGION Network 2: Anforderung zum Ausführen der Funktion
   RUNG wire#powerrail
      Contact( "allgDataTestSendRcvIJaw".xTriggerStartIsduAuftrag )
      wire#w1
      Coil( "allgDataTestSendRcvIJaw".udtFreeIsduCmd.execute )
   END_RUNG
   RUNG wire#w1
      Contact( #READ_WRITE_ISDU_CMD_GAIN )
      Move(in := #WRITE_LENGTH_ISDU_CMD_GAIN, out1 => "allgDataTestSendRcvIJaw".udtFreeIsduCmd.writeLen)
      Coil( "allgDataTestSendRcvIJaw".udtFreeIsduCmd.readWrite )
   END_RUNG
   RUNG wire#w1
      Move(in := #IDX_IJAW_1, out1 => "allgDataTestSendRcvIJaw".udtFreeIsduCmd.port)
   END_RUNG
   RUNG wire#w1
      Move(in := #IDX_ISDU_CMD_GAIN, out1 => "allgDataTestSendRcvIJaw".udtFreeIsduCmd.index)
   END_RUNG
   RUNG wire#w1
      Move(in := #SUB_IDX_ISDU_CMD_GAIN, out1 => "allgDataTestSendRcvIJaw".udtFreeIsduCmd.subindex)
   END_RUNG
   // the same network as SCL:
   "allgDataTestSendRcvIJaw".udtFreeIsduCmd.execute := "allgDataTestSendRcvIJaw".xTriggerStartIsduAuftrag;
   #_w1 := "allgDataTestSendRcvIJaw".xTriggerStartIsduAuftrag AND #READ_WRITE_ISDU_CMD_GAIN;
   IF #_w1 THEN "allgDataTestSendRcvIJaw".udtFreeIsduCmd.writeLen := #WRITE_LENGTH_ISDU_CMD_GAIN; END_IF;
   "allgDataTestSendRcvIJaw".udtFreeIsduCmd.readWrite := #_w1;
   IF "allgDataTestSendRcvIJaw".xTriggerStartIsduAuftrag THEN
       "allgDataTestSendRcvIJaw".udtFreeIsduCmd.port := #IDX_IJAW_1;
       "allgDataTestSendRcvIJaw".udtFreeIsduCmd.index := #IDX_ISDU_CMD_GAIN;
       "allgDataTestSendRcvIJaw".udtFreeIsduCmd.subindex := #SUB_IDX_ISDU_CMD_GAIN;
   END_IF;
END_REGION

REGION Network 3: CALL SEN / RCV IJAW DATA 8-PORT
   // "TigoMaster2TH~IODevice" --> 8 Port Device
   // 
   // Folgendes kann an iLADDRR_TigoMaster parametriert werden: 
   // - #hwDeviceTigoMaster (siehe Netzwerk 1)
   // - "TigoMaster2TH~IODevice" (abhängig vom Namen des TigoMasters in der Hardwarekonfiguration)
   // - 281 (anhängig des Wertes der Systemkonstante "TigoMaster2TH~IODevice")
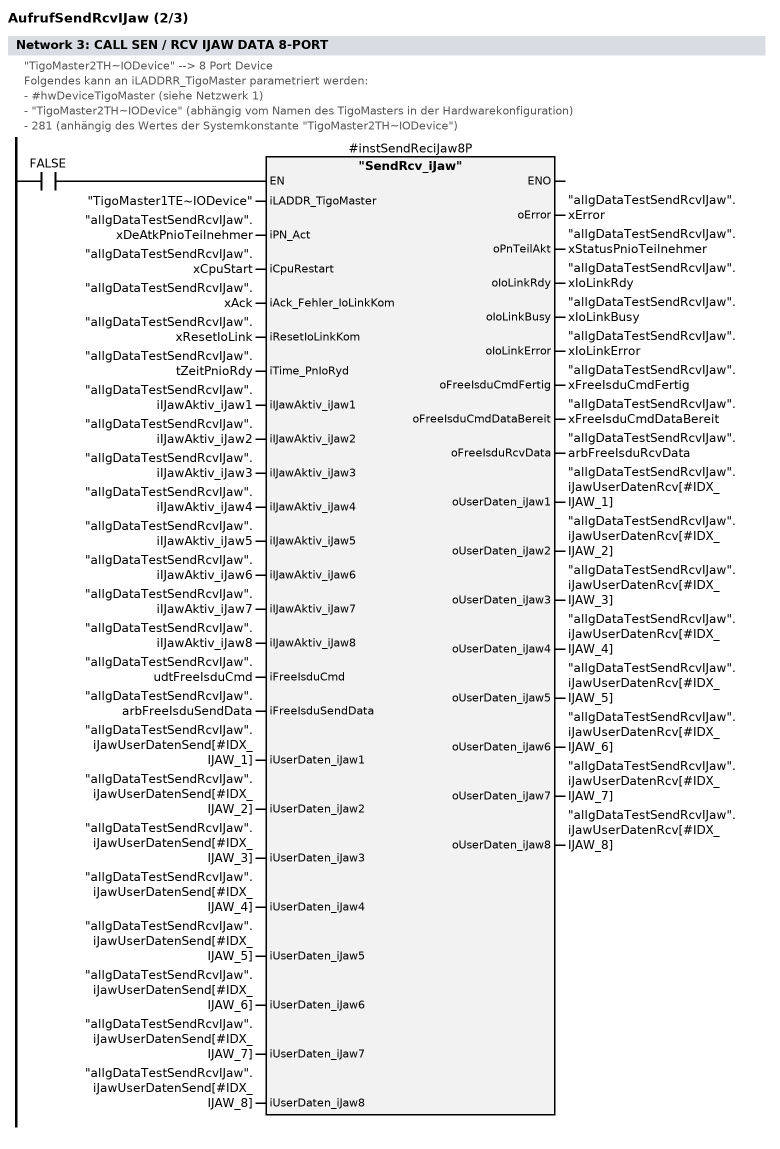
   RUNG wire#powerrail
      Contact( FALSE )
      #instSendReciJaw8P(iLADDR_TigoMaster := "TigoMaster1TE~IODevice", iPN_Act := "allgDataTestSendRcvIJaw".xDeAtkPnioTeilnehmer, iCpuRestart := "allgDataTestSendRcvIJaw".xCpuStart, iAck_Fehler_IoLinkKom := "allgDataTestSendRcvIJaw".xAck, iResetIoLinkKom := "allgDataTestSendRcvIJaw".xResetIoLink, iTime_PnIoRyd := "allgDataTestSendRcvIJaw".tZeitPnioRdy, iIJawAktiv_iJaw1 := "allgDataTestSendRcvIJaw".iIJawAktiv_iJaw1, iIJawAktiv_iJaw2 := "allgDataTestSendRcvIJaw".iIJawAktiv_iJaw2, iIJawAktiv_iJaw3 := "allgDataTestSendRcvIJaw".iIJawAktiv_iJaw3, iIJawAktiv_iJaw4 := "allgDataTestSendRcvIJaw".iIJawAktiv_iJaw4, iIJawAktiv_iJaw5 := "allgDataTestSendRcvIJaw".iIJawAktiv_iJaw5, iIJawAktiv_iJaw6 := "allgDataTestSendRcvIJaw".iIJawAktiv_iJaw6, iIJawAktiv_iJaw7 := "allgDataTestSendRcvIJaw".iIJawAktiv_iJaw7, iIJawAktiv_iJaw8 := "allgDataTestSendRcvIJaw".iIJawAktiv_iJaw8, iFreeIsduCmd := "allgDataTestSendRcvIJaw".udtFreeIsduCmd, iFreeIsduSendData := "allgDataTestSendRcvIJaw".arbFreeIsduSendData, iUserDaten_iJaw1 := "allgDataTestSendRcvIJaw".iJawUserDatenSend[#IDX_IJAW_1], iUserDaten_iJaw2 := "allgDataTestSendRcvIJaw".iJawUserDatenSend[#IDX_IJAW_2], iUserDaten_iJaw3 := "allgDataTestSendRcvIJaw".iJawUserDatenSend[#IDX_IJAW_3], iUserDaten_iJaw4 := "allgDataTestSendRcvIJaw".iJawUserDatenSend[#IDX_IJAW_4], iUserDaten_iJaw5 := "allgDataTestSendRcvIJaw".iJawUserDatenSend[#IDX_IJAW_5], iUserDaten_iJaw6 := "allgDataTestSendRcvIJaw".iJawUserDatenSend[#IDX_IJAW_6], iUserDaten_iJaw7 := "allgDataTestSendRcvIJaw".iJawUserDatenSend[#IDX_IJAW_7], iUserDaten_iJaw8 := "allgDataTestSendRcvIJaw".iJawUserDatenSend[#IDX_IJAW_8], oError => "allgDataTestSendRcvIJaw".xError, oPnTeilAkt => "allgDataTestSendRcvIJaw".xStatusPnioTeilnehmer, oIoLinkRdy => "allgDataTestSendRcvIJaw".xIoLinkRdy, oIoLinkBusy => "allgDataTestSendRcvIJaw".xIoLinkBusy, oIoLinkError => "allgDataTestSendRcvIJaw".xIoLinkError, oFreeIsduCmdFertig => "allgDataTestSendRcvIJaw".xFreeIsduCmdFertig, oFreeIsduCmdDataBereit => "allgDataTestSendRcvIJaw".xFreeIsduCmdDataBereit, oFreeIsduRcvData => "allgDataTestSendRcvIJaw".arbFreeIsduRcvData, oUserDaten_iJaw1 => "allgDataTestSendRcvIJaw".iJawUserDatenRcv[#IDX_IJAW_1], oUserDaten_iJaw2 => "allgDataTestSendRcvIJaw".iJawUserDatenRcv[#IDX_IJAW_2], oUserDaten_iJaw3 => "allgDataTestSendRcvIJaw".iJawUserDatenRcv[#IDX_IJAW_3], oUserDaten_iJaw4 => "allgDataTestSendRcvIJaw".iJawUserDatenRcv[#IDX_IJAW_4], oUserDaten_iJaw5 => "allgDataTestSendRcvIJaw".iJawUserDatenRcv[#IDX_IJAW_5], oUserDaten_iJaw6 => "allgDataTestSendRcvIJaw".iJawUserDatenRcv[#IDX_IJAW_6], oUserDaten_iJaw7 => "allgDataTestSendRcvIJaw".iJawUserDatenRcv[#IDX_IJAW_7], oUserDaten_iJaw8 => "allgDataTestSendRcvIJaw".iJawUserDatenRcv[#IDX_IJAW_8])
   END_RUNG
   // the same network as SCL:
   IF FALSE THEN
       #instSendReciJaw8P(iLADDR_TigoMaster := "TigoMaster1TE~IODevice",   // "SendRcv_iJaw"
                          iPN_Act := "allgDataTestSendRcvIJaw".xDeAtkPnioTeilnehmer,
                          iCpuRestart := "allgDataTestSendRcvIJaw".xCpuStart,
                          iAck_Fehler_IoLinkKom := "allgDataTestSendRcvIJaw".xAck,
                          iResetIoLinkKom := "allgDataTestSendRcvIJaw".xResetIoLink,
                          iTime_PnIoRyd := "allgDataTestSendRcvIJaw".tZeitPnioRdy,
                          iIJawAktiv_iJaw1 := "allgDataTestSendRcvIJaw".iIJawAktiv_iJaw1,
                          iIJawAktiv_iJaw2 := "allgDataTestSendRcvIJaw".iIJawAktiv_iJaw2,
                          iIJawAktiv_iJaw3 := "allgDataTestSendRcvIJaw".iIJawAktiv_iJaw3,
                          iIJawAktiv_iJaw4 := "allgDataTestSendRcvIJaw".iIJawAktiv_iJaw4,
                          iIJawAktiv_iJaw5 := "allgDataTestSendRcvIJaw".iIJawAktiv_iJaw5,
                          iIJawAktiv_iJaw6 := "allgDataTestSendRcvIJaw".iIJawAktiv_iJaw6,
                          iIJawAktiv_iJaw7 := "allgDataTestSendRcvIJaw".iIJawAktiv_iJaw7,
                          iIJawAktiv_iJaw8 := "allgDataTestSendRcvIJaw".iIJawAktiv_iJaw8,
                          iFreeIsduCmd := "allgDataTestSendRcvIJaw".udtFreeIsduCmd,
                          iFreeIsduSendData := "allgDataTestSendRcvIJaw".arbFreeIsduSendData,
                          iUserDaten_iJaw1 := "allgDataTestSendRcvIJaw".iJawUserDatenSend[#IDX_IJAW_1],
                          iUserDaten_iJaw2 := "allgDataTestSendRcvIJaw".iJawUserDatenSend[#IDX_IJAW_2],
                          iUserDaten_iJaw3 := "allgDataTestSendRcvIJaw".iJawUserDatenSend[#IDX_IJAW_3],
                          iUserDaten_iJaw4 := "allgDataTestSendRcvIJaw".iJawUserDatenSend[#IDX_IJAW_4],
                          iUserDaten_iJaw5 := "allgDataTestSendRcvIJaw".iJawUserDatenSend[#IDX_IJAW_5],
                          iUserDaten_iJaw6 := "allgDataTestSendRcvIJaw".iJawUserDatenSend[#IDX_IJAW_6],
                          iUserDaten_iJaw7 := "allgDataTestSendRcvIJaw".iJawUserDatenSend[#IDX_IJAW_7],
                          iUserDaten_iJaw8 := "allgDataTestSendRcvIJaw".iJawUserDatenSend[#IDX_IJAW_8],
                          oError => "allgDataTestSendRcvIJaw".xError,
                          oPnTeilAkt => "allgDataTestSendRcvIJaw".xStatusPnioTeilnehmer,
                          oIoLinkRdy => "allgDataTestSendRcvIJaw".xIoLinkRdy,
                          oIoLinkBusy => "allgDataTestSendRcvIJaw".xIoLinkBusy,
                          oIoLinkError => "allgDataTestSendRcvIJaw".xIoLinkError,
                          oFreeIsduCmdFertig => "allgDataTestSendRcvIJaw".xFreeIsduCmdFertig,
                          oFreeIsduCmdDataBereit => "allgDataTestSendRcvIJaw".xFreeIsduCmdDataBereit,
                          oFreeIsduRcvData => "allgDataTestSendRcvIJaw".arbFreeIsduRcvData,
                          oUserDaten_iJaw1 => "allgDataTestSendRcvIJaw".iJawUserDatenRcv[#IDX_IJAW_1],
                          oUserDaten_iJaw2 => "allgDataTestSendRcvIJaw".iJawUserDatenRcv[#IDX_IJAW_2],
                          oUserDaten_iJaw3 => "allgDataTestSendRcvIJaw".iJawUserDatenRcv[#IDX_IJAW_3],
                          oUserDaten_iJaw4 => "allgDataTestSendRcvIJaw".iJawUserDatenRcv[#IDX_IJAW_4],
                          oUserDaten_iJaw5 => "allgDataTestSendRcvIJaw".iJawUserDatenRcv[#IDX_IJAW_5],
                          oUserDaten_iJaw6 => "allgDataTestSendRcvIJaw".iJawUserDatenRcv[#IDX_IJAW_6],
                          oUserDaten_iJaw7 => "allgDataTestSendRcvIJaw".iJawUserDatenRcv[#IDX_IJAW_7],
                          oUserDaten_iJaw8 => "allgDataTestSendRcvIJaw".iJawUserDatenRcv[#IDX_IJAW_8]);
   END_IF;
END_REGION

REGION Network 4: CALL SEN / RCV IJAW DATA 4-PORT
   // "TigoMaster1TE~IODevice" --> 4 Port Device
   // 
   // Folgendes kann an iLADDRR_TigoMaster parametriert werden: 
   // - #hwDeviceTigoMaster (siehe Netzwerk 1)
   // - "TigoMaster2TH~IODevice" (abhängig vom Namen des TigoMasters in der Hardwarekonfiguration)
   // - 281 (anhängig des Wertes der Systemkonstante "TigoMaster2TH~IODevice")
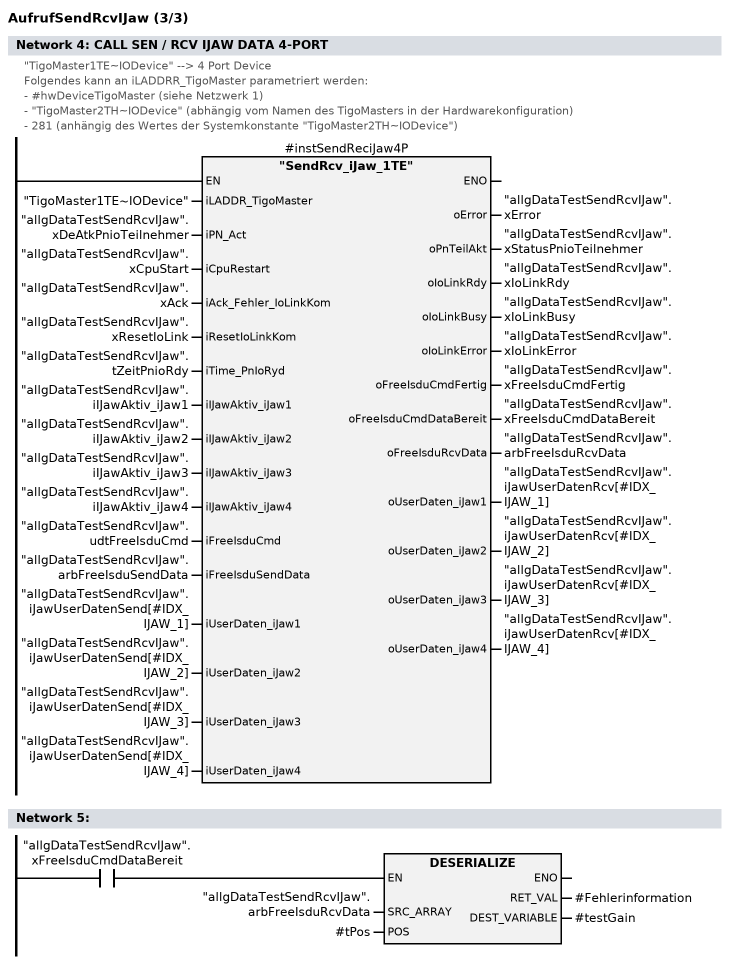
   RUNG wire#powerrail
      #instSendReciJaw4P(iLADDR_TigoMaster := "TigoMaster1TE~IODevice", iPN_Act := "allgDataTestSendRcvIJaw".xDeAtkPnioTeilnehmer, iCpuRestart := "allgDataTestSendRcvIJaw".xCpuStart, iAck_Fehler_IoLinkKom := "allgDataTestSendRcvIJaw".xAck, iResetIoLinkKom := "allgDataTestSendRcvIJaw".xResetIoLink, iTime_PnIoRyd := "allgDataTestSendRcvIJaw".tZeitPnioRdy, iIJawAktiv_iJaw1 := "allgDataTestSendRcvIJaw".iIJawAktiv_iJaw1, iIJawAktiv_iJaw2 := "allgDataTestSendRcvIJaw".iIJawAktiv_iJaw2, iIJawAktiv_iJaw3 := "allgDataTestSendRcvIJaw".iIJawAktiv_iJaw3, iIJawAktiv_iJaw4 := "allgDataTestSendRcvIJaw".iIJawAktiv_iJaw4, iFreeIsduCmd := "allgDataTestSendRcvIJaw".udtFreeIsduCmd, iFreeIsduSendData := "allgDataTestSendRcvIJaw".arbFreeIsduSendData, iUserDaten_iJaw1 := "allgDataTestSendRcvIJaw".iJawUserDatenSend[#IDX_IJAW_1], iUserDaten_iJaw2 := "allgDataTestSendRcvIJaw".iJawUserDatenSend[#IDX_IJAW_2], iUserDaten_iJaw3 := "allgDataTestSendRcvIJaw".iJawUserDatenSend[#IDX_IJAW_3], iUserDaten_iJaw4 := "allgDataTestSendRcvIJaw".iJawUserDatenSend[#IDX_IJAW_4], oError => "allgDataTestSendRcvIJaw".xError, oPnTeilAkt => "allgDataTestSendRcvIJaw".xStatusPnioTeilnehmer, oIoLinkRdy => "allgDataTestSendRcvIJaw".xIoLinkRdy, oIoLinkBusy => "allgDataTestSendRcvIJaw".xIoLinkBusy, oIoLinkError => "allgDataTestSendRcvIJaw".xIoLinkError, oFreeIsduCmdFertig => "allgDataTestSendRcvIJaw".xFreeIsduCmdFertig, oFreeIsduCmdDataBereit => "allgDataTestSendRcvIJaw".xFreeIsduCmdDataBereit, oFreeIsduRcvData => "allgDataTestSendRcvIJaw".arbFreeIsduRcvData, oUserDaten_iJaw1 => "allgDataTestSendRcvIJaw".iJawUserDatenRcv[#IDX_IJAW_1], oUserDaten_iJaw2 => "allgDataTestSendRcvIJaw".iJawUserDatenRcv[#IDX_IJAW_2], oUserDaten_iJaw3 => "allgDataTestSendRcvIJaw".iJawUserDatenRcv[#IDX_IJAW_3], oUserDaten_iJaw4 => "allgDataTestSendRcvIJaw".iJawUserDatenRcv[#IDX_IJAW_4])
   END_RUNG
   // the same network as SCL:
   #instSendReciJaw4P(iLADDR_TigoMaster := "TigoMaster1TE~IODevice",   // "SendRcv_iJaw_1TE"
                      iPN_Act := "allgDataTestSendRcvIJaw".xDeAtkPnioTeilnehmer,
                      iCpuRestart := "allgDataTestSendRcvIJaw".xCpuStart,
                      iAck_Fehler_IoLinkKom := "allgDataTestSendRcvIJaw".xAck,
                      iResetIoLinkKom := "allgDataTestSendRcvIJaw".xResetIoLink,
                      iTime_PnIoRyd := "allgDataTestSendRcvIJaw".tZeitPnioRdy,
                      iIJawAktiv_iJaw1 := "allgDataTestSendRcvIJaw".iIJawAktiv_iJaw1,
                      iIJawAktiv_iJaw2 := "allgDataTestSendRcvIJaw".iIJawAktiv_iJaw2,
                      iIJawAktiv_iJaw3 := "allgDataTestSendRcvIJaw".iIJawAktiv_iJaw3,
                      iIJawAktiv_iJaw4 := "allgDataTestSendRcvIJaw".iIJawAktiv_iJaw4,
                      iFreeIsduCmd := "allgDataTestSendRcvIJaw".udtFreeIsduCmd,
                      iFreeIsduSendData := "allgDataTestSendRcvIJaw".arbFreeIsduSendData,
                      iUserDaten_iJaw1 := "allgDataTestSendRcvIJaw".iJawUserDatenSend[#IDX_IJAW_1],
                      iUserDaten_iJaw2 := "allgDataTestSendRcvIJaw".iJawUserDatenSend[#IDX_IJAW_2],
                      iUserDaten_iJaw3 := "allgDataTestSendRcvIJaw".iJawUserDatenSend[#IDX_IJAW_3],
                      iUserDaten_iJaw4 := "allgDataTestSendRcvIJaw".iJawUserDatenSend[#IDX_IJAW_4],
                      oError => "allgDataTestSendRcvIJaw".xError,
                      oPnTeilAkt => "allgDataTestSendRcvIJaw".xStatusPnioTeilnehmer,
                      oIoLinkRdy => "allgDataTestSendRcvIJaw".xIoLinkRdy,
                      oIoLinkBusy => "allgDataTestSendRcvIJaw".xIoLinkBusy,
                      oIoLinkError => "allgDataTestSendRcvIJaw".xIoLinkError,
                      oFreeIsduCmdFertig => "allgDataTestSendRcvIJaw".xFreeIsduCmdFertig,
                      oFreeIsduCmdDataBereit => "allgDataTestSendRcvIJaw".xFreeIsduCmdDataBereit,
                      oFreeIsduRcvData => "allgDataTestSendRcvIJaw".arbFreeIsduRcvData,
                      oUserDaten_iJaw1 => "allgDataTestSendRcvIJaw".iJawUserDatenRcv[#IDX_IJAW_1],
                      oUserDaten_iJaw2 => "allgDataTestSendRcvIJaw".iJawUserDatenRcv[#IDX_IJAW_2],
                      oUserDaten_iJaw3 => "allgDataTestSendRcvIJaw".iJawUserDatenRcv[#IDX_IJAW_3],
                      oUserDaten_iJaw4 => "allgDataTestSendRcvIJaw".iJawUserDatenRcv[#IDX_IJAW_4]);
END_REGION

REGION Network 5
   // no SCL statement known for Deserialize: written as a call
   IF "allgDataTestSendRcvIJaw".xFreeIsduCmdDataBereit THEN
       #Fehlerinformation := Deserialize(SRC_ARRAY := "allgDataTestSendRcvIJaw".arbFreeIsduRcvData,
                               POS := #tPos,
                               DEST_VARIABLE => #testGain);
   END_IF;
END_REGION
END_FUNCTION_BLOCK

// ===== library: MasterCopy "allgDataTestSendRcvIJaw" =====

DATA_BLOCK "allgDataTestSendRcvIJaw"   // DB2
{ S7_Optimized_Access := 'TRUE' }
VERSION : 0.1
   VAR
      xCpuStart : Bool := FALSE;   // erster zyklus nach cpu start
      xDeAtkPnioTeilnehmer : Bool;   // De-/Aktivierung Profinetteilnehmer 1= Aktivieren 0= Deaktivieren
      xError : Bool;   // Fehler bei der Abarbeitung des Bausteines
      xStatusPnioTeilnehmer : Bool;   // Status des Profinetteilnehmer 1= Teilnehmer aktiv 0= Teilnehmer deaktiviert
      xAck : Bool;   // Quitterung des Kommunikationsfehlers.(Sende-/ Lese Aufträge werden danach erneut gestartet)
      xResetIoLink : Bool;   // Reset der LIO-Link kommunikation (Alle Sende-/ Lese Aufträge werden gelöscht)
      tZeitPnioRdy : Time := T#5s;   // Zeit zum Hochlauf des Bussystems / des TigoMasters (Vermeidung von Lesefehlern)
      iIJawAktiv_iJaw1 : Bool := TRUE;   // iJaw 1 ist aktiv & vorhanden
      iIJawAktiv_iJaw2 : Bool;   // iJaw 2 ist aktiv & vorhanden
      iIJawAktiv_iJaw3 : Bool;   // iJaw 3 ist aktiv & vorhanden
      iIJawAktiv_iJaw4 : Bool;   // iJaw 4 ist aktiv & vorhanden
      iIJawAktiv_iJaw5 : Bool;   // iJaw 5 ist aktiv & vorhanden
      iIJawAktiv_iJaw6 : Bool;   // iJaw 6 ist aktiv & vorhanden
      iIJawAktiv_iJaw7 : Bool;   // iJaw 7 ist aktiv & vorhanden
      iIJawAktiv_iJaw8 : Bool;   // iJaw 7 ist aktiv & vorhanden
      xIoLinkRdy : Bool;   // Ío link kommunikation bereit zum senden / empfangen
      xIoLinkBusy : Bool;   // Ío link kommunikation beschäftig
      xIoLinkError : Bool;   // Ío link kommunikation fehlerhaft
      xFreeIsduCmdFertig : Bool;   // Freier ISDU-Auftrag erfolgreich abgeschlossen
      xFreeIsduCmdDataBereit : Bool;   // Empfange ISDU-Daten liegen bereit
      xTriggerStartIsduAuftrag : Bool;   // Freier Trigger starte Isdu-Auftrag
      udtFreeIsduCmd : "UDT_iJawISDUCmdData";   // Freier ISDU-Auftrag
      arbFreeIsduSendData : Array[0..231] of Byte;   // Datenbereich zum Schreiben für den freien ISDU-Auftrag
      arbFreeIsduRcvData : Array[0..231] of Byte;   // Datenbereich zum Schreiben für den freien ISDU-Auftrag
      iJawUserDatenSend : Array[1..8] of "UDT_iJawDataSendUser";   // Daten / Befehle welche an den Tigomaster gesendet werden
      iJawUserDatenRcv : Array[1..8] of "UDT_iJawDataRcvUser";   // Daten welche vom Tigomaster gelesen werden
   END_VAR
BEGIN
   // udtFreeIsduCmd.port : Port am IO-Link-Master-Modul (Nummer der iJaw 1-8)
END_DATA_BLOCK

// ===== library: MasterCopy "AufrufSendRcvIJaw_DB" =====

DATA_BLOCK "AufrufSendRcvIJaw_DB"   // DB1
{ S7_Optimized_Access := 'TRUE' }
VERSION : 0.1
// stored: InstanceOfName AufrufSendRcvIJaw
"AufrufSendRcvIJaw"
BEGIN
END_DATA_BLOCK